TYPE S_User_Data :
STRUCT
	UserData AT %Q* : ARRAY [0..63] OF BYTE;
END_STRUCT
END_TYPE

(* stored: Version 1.1.0.1, ProductVersion 3.1.4024.10
   DUT S_User_Data: Id {20e842b5-31eb-40de-94d4-e35e96147b74} *)
